VAR_GLOBAL CONSTANT
	cRECVDATACHANNELBUFFER 		:INT := 20;
END_VAR

(* stored: Version 1.1.0.1, ProductVersion 3.1.0.24
   GVL IdBaseConst: Id {cb0632dc-c560-4fd5-9cb8-e5f3818cb927} *)
